SYSTEM TEST_NW (* Test of Network Segments and Links *)
  (* Standard: 61499-1 *)
  (* Version 0.0, 2004-02-21, JHC, Rockwell Automation *)
  DEVICE DEV1 : FRAME_DEVICE(BOUNDS := [0,0,0,0])
    RESOURCE RES2 : PANEL_RESOURCE(ROWS := 0)
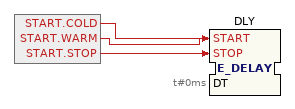
      FBS
        DLY : E_DELAY(DT := t#0ms);
      END_FBS
      EVENT_CONNECTIONS
        START.COLD TO DLY.START;
        START.WARM TO DLY.START;
        START.STOP TO DLY.STOP;
      END_CONNECTIONS
    END_RESOURCE
  END_DEVICE
  DEVICE PLC1 : RMT_DEV
  END_DEVICE
  DEVICE PLC2 : RMT_DEV
  END_DEVICE
  DEVICE IO1 : RMT_DEV
  END_DEVICE
  DEVICE IO2 : RMT_DEV
  END_DEVICE
  DEVICE DEV2 : FRAME_DEVICE
  END_DEVICE
  SEGMENTS
    SEG1 : Ethernet(SPEED := 100Mbps (* A parameter comment *), LENGTH := 100m (* Another parameter comment *)); (* A Segment Comment *)
    SEG2 : DeviceNet(SPEED := 500Kbps);
    SEG3 : LocalBus; (* Test segment with comment but no parameters *)
  END_SEGMENTS
  LINKS
    DEV1 => SEG1(TYPE := ThinWire (* A link parameter comment *), LENGTH := 500mm (* Another one *)); (* A link comment *)
    PLC1 => SEG1;
    PLC2 => SEG1;
    PLC2 => SEG2;
    IO1 => SEG2(LENGTH := 100mm);
    IO2 => SEG2(LENGTH := 50mm);
    DEV1 => SEG3;
    DEV2 => SEG3;
  END_LINKS
END_SYSTEM
